// TIA Portal V16 program export: 1 tag tables, 0 data types, 1 data blocks, 2 code blocks (in call order from the OBs), 2 instance data blocks

VAR_GLOBAL   // PLC tag table "Default tag table"
   Clock_Byte AT %MB0 : Byte;
   Clock_10Hz AT %M0.0 : Bool;
   Clock_5Hz AT %M0.1 : Bool;
   "Clock_2.5Hz" AT %M0.2 : Bool;
   Clock_2Hz AT %M0.3 : Bool;
   "Clock_1.25Hz" AT %M0.4 : Bool;
   Clock_1Hz AT %M0.5 : Bool;
   "Clock_0.625Hz" AT %M0.6 : Bool;
   "Clock_0.5Hz" AT %M0.7 : Bool;
   "Disconect request" AT %M1.0 : Bool;
   "Send on/off" AT %M1.1 : Bool;
   "Receive enable" AT %M1.2 : Bool;
   "mine-tag" AT %M1.3 : Bool;
   nuevo_tag AT %M1.4 : Bool;
END_VAR

DATA_BLOCK "DATA"   // DB6
{ S7_Optimized_Access := 'TRUE' }
VERSION : 0.1
// stored: AutoNumber true, IsOnlyStoredInLoadMemory false, IsRetainMemResEnabled false, IsWriteProtectedInAS false, MemoryReserve 100
   VAR
      Receive : Array[0..20] of Char;
      Send : String := 'Hello world!';
      Do_Connect : Bool;
      Passive_Conn_Done : Bool;
   END_VAR
BEGIN
END_DATA_BLOCK

ORGANIZATION_BLOCK "Main"   // OB1, LAD, ProgramCycle
TITLE = "Main Program Sweep (Cycle)"
{ S7_Optimized_Access := 'TRUE' }
VERSION : 0.1
// stored: AutoNumber true, IsIECCheckEnabled false, SetENOAutomatically false
   VAR_INPUT
      Initial_Call : Bool;   // Initial call of this OB
      Remanence : Bool;   // =True, if remanent data are available
   END_VAR
   VAR_TEMP
      suma : Int;
   END_VAR
BEGIN

REGION Network 1
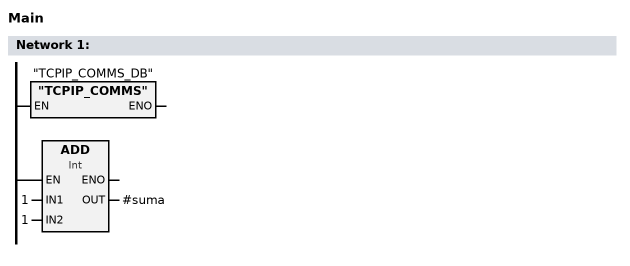
   RUNG wire#powerrail
      "TCPIP_COMMS_DB"()
   END_RUNG
   RUNG wire#powerrail
      { S7_Templates := "SrcType := Int" } Add(in1 := 1, in2 := 1, out => #suma)
   END_RUNG
   // the same network as SCL:
   "TCPIP_COMMS_DB"();   // "TCPIP_COMMS"
   #suma := 1 + 1;
END_REGION
END_ORGANIZATION_BLOCK

FUNCTION_BLOCK "TCPIP_COMMS"   // FB1, LAD
{ S7_Optimized_Access := 'TRUE' }
VERSION : 0.1
// stored: AutoNumber true, IsIECCheckEnabled false, IsRetainMemResEnabled false, MemoryReserve 100, SetENOAutomatically false, UDAEnableTagReadback false
   VAR
      TCON : Struct
         REQ : Bool;
         DONE : Bool;
         BUSY : Bool;
         ERROR : Bool;
         STATUS : UInt;
         DONESAVE : Bool;
      END_STRUCT;
      TDISCON : Struct
         REQ : Bool;
         DONE : Bool;
         BUSY : Bool;
         ERROR : Bool;
         DONESAVE : Bool;
         STATUS : UInt;
      END_STRUCT;
      TSEND : Struct
         REQ : Bool;
         DONE : Bool;
         BUSY : Bool;
         ERROR : Bool;
         DONESAVE : Bool;
         STATUS : UInt;
      END_STRUCT;
      TRCV : Struct
         EN_R : Bool;
         NDR : Bool;
         BUSY : Bool;
         ERROR : Bool;
         STATUS : UInt;
         RCVD_LEN : UDInt;
      END_STRUCT;
      ReceivedString : String;
      TCON_DB { ExternalAccessible := 'False'; ExternalVisible := 'False'; ExternalWritable := 'False'} : TCON;
      TDISCON_DB { ExternalAccessible := 'False'; ExternalVisible := 'False'; ExternalWritable := 'False'} : TDISCON;
      TSEND_DB { ExternalAccessible := 'False'; ExternalVisible := 'False'; ExternalWritable := 'False'} : TSEND;
      TRCV_DB { ExternalAccessible := 'False'; ExternalVisible := 'False'; ExternalWritable := 'False'} : TRCV;
   END_VAR
BEGIN

REGION Network 1: TCON
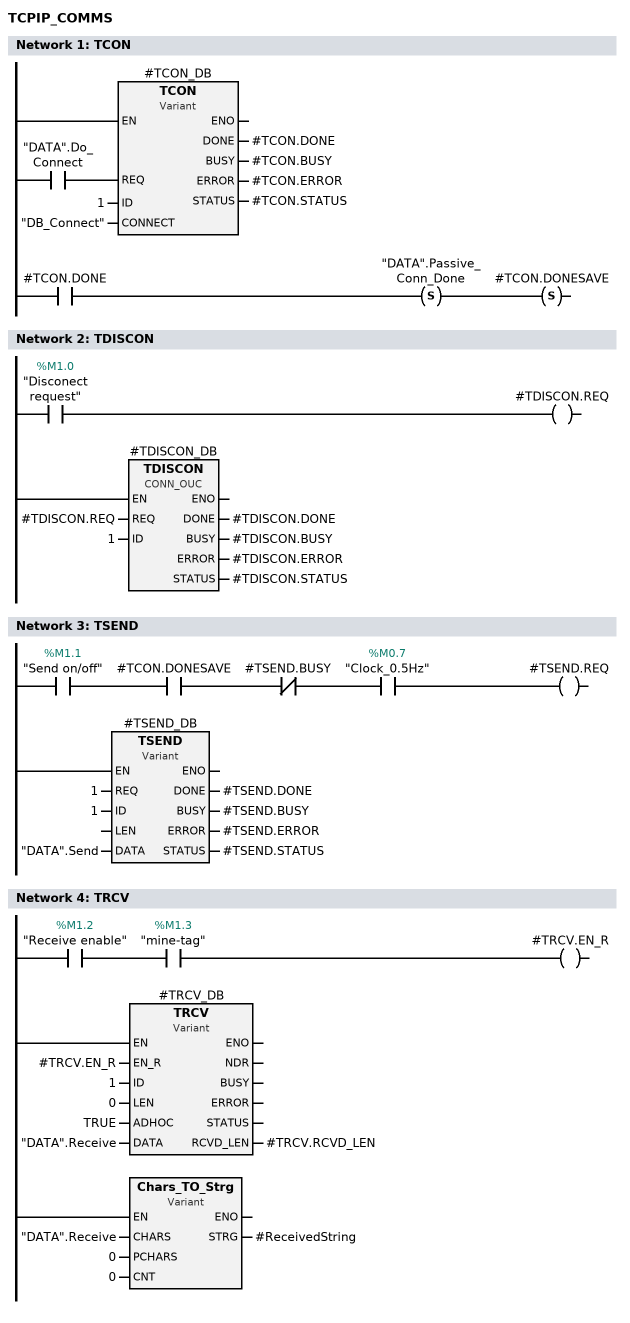
   RUNG wire#powerrail
      { S7_Templates := "[con_type := Variant, id_type := CONN_OUC]" } #TCON_DB.TCON(REQ := wire#w1, ID := 1, CONNECT := "DB_Connect", DONE => #TCON.DONE, BUSY => #TCON.BUSY, ERROR => #TCON.ERROR, STATUS => #TCON.STATUS)
   END_RUNG
   RUNG wire#powerrail
      Contact( "DATA".Do_Connect )
   END_RUNG wire#w1
   RUNG wire#powerrail
      Contact( #TCON.DONE )
      S_Coil( "DATA".Passive_Conn_Done )
      S_Coil( #TCON.DONESAVE )
   END_RUNG
   // the same network as SCL:
   #TCON_DB(REQ := "DATA".Do_Connect,   // TCON
            ID := 1,
            CONNECT := "DB_Connect",
            DONE => #TCON.DONE,
            BUSY => #TCON.BUSY,
            ERROR => #TCON.ERROR,
            STATUS => #TCON.STATUS);
   IF #TCON.DONE THEN
       "DATA".Passive_Conn_Done := TRUE;
       #TCON.DONESAVE := TRUE;
   END_IF;
END_REGION

REGION Network 2: TDISCON
   RUNG wire#powerrail
      Contact( "Disconect request" )
      Coil( #TDISCON.REQ )
   END_RUNG
   RUNG wire#powerrail
      { S7_Templates := "id_type := CONN_OUC" } #TDISCON_DB.TDISCON(REQ := #TDISCON.REQ, ID := 1, DONE => #TDISCON.DONE, BUSY => #TDISCON.BUSY, ERROR => #TDISCON.ERROR, STATUS => #TDISCON.STATUS)
   END_RUNG
   // the same network as SCL:
   #TDISCON.REQ := "Disconect request";
   #TDISCON_DB(REQ := #TDISCON.REQ,   // TDISCON
               ID := 1,
               DONE => #TDISCON.DONE,
               BUSY => #TDISCON.BUSY,
               ERROR => #TDISCON.ERROR,
               STATUS => #TDISCON.STATUS);
END_REGION

REGION Network 3: TSEND
   RUNG wire#powerrail
      Contact( "Send on/off" )
      Contact( #TCON.DONESAVE )
      I_Contact( #TSEND.BUSY )
      Contact( "Clock_0.5Hz" )
      Coil( #TSEND.REQ )
   END_RUNG
   RUNG wire#powerrail
      { S7_Templates := "[data_type := Variant, len_type := UDInt, id_type := CONN_OUC]" } #TSEND_DB.TSEND(REQ := 1, ID := 1, LEN :=, DATA := "DATA".Send, DONE => #TSEND.DONE, BUSY => #TSEND.BUSY, ERROR => #TSEND.ERROR, STATUS => #TSEND.STATUS)
   END_RUNG
   // the same network as SCL:
   #TSEND.REQ := "Send on/off" AND #TCON.DONESAVE AND NOT #TSEND.BUSY AND "Clock_0.5Hz";
   #TSEND_DB(REQ := 1,   // TSEND
             ID := 1,
             DATA := "DATA".Send,
             DONE => #TSEND.DONE,
             BUSY => #TSEND.BUSY,
             ERROR => #TSEND.ERROR,
             STATUS => #TSEND.STATUS);
END_REGION

REGION Network 4: TRCV
   RUNG wire#powerrail
      Contact( "Receive enable" )
      Contact( "mine-tag" )
      Coil( #TRCV.EN_R )
   END_RUNG
   RUNG wire#powerrail
      { S7_Templates := "[card := 1, ptr_type := Variant, value_type := UDInt, id_type := CONN_OUC]" } #TRCV_DB.TRCV(EN_R := #TRCV.EN_R, ID := 1, LEN := 0, ADHOC := TRUE, DATA := "DATA".Receive, NDR =>, BUSY =>, ERROR =>, STATUS =>, RCVD_LEN => #TRCV.RCVD_LEN)
   END_RUNG
   RUNG wire#powerrail
      { S7_Templates := "[ptr_type := Variant, str_type := String]" } Chars_TO_Strg(Chars := "DATA".Receive, pChars := 0, Cnt := 0, Strg => #ReceivedString)
   END_RUNG
   // the same network as SCL:
   #TRCV.EN_R := "Receive enable" AND "mine-tag";
   #TRCV_DB(EN_R := #TRCV.EN_R,   // TRCV
            ID := 1,
            LEN := 0,
            ADHOC := TRUE,
            DATA := "DATA".Receive,
            RCVD_LEN => #TRCV.RCVD_LEN);
   Chars_TO_Strg(Chars := "DATA".Receive, pChars := 0, Cnt := 0, Strg => #ReceivedString);
END_REGION
END_FUNCTION_BLOCK

DATA_BLOCK "TCPIP_COMMS_DB"   // DB1
VERSION : 0.1
// stored: AutoNumber true, InstanceOfName TCPIP_COMMS, InstanceOfType FB
"TCPIP_COMMS"
BEGIN
END_DATA_BLOCK

DATA_BLOCK "DB_Connect"   // DB2
{ S7_Optimized_Access := 'TRUE' }
// stored: AutoNumber true, InstanceOfName TCON_IP_v4, OfSystemLibElement TCON_IP_v4, OfSystemLibVersion 1.0
"TCON_IP_v4"
   // VAR
   //    InterfaceId : HW_ANY := 64;
   //    ID : CONN_OUC := 1;
   //    ConnectionType : Byte;
   //    ActiveEstablished : Bool := false;
   //    RemoteAddress { S7_SetPoint := 'True'} : IP_V4;
   //    RemotePort : UInt := 0;
   //    LocalPort : UInt := 5000;
   // END_VAR
BEGIN
   RemoteAddress.ADDR[1] := 192;
   RemoteAddress.ADDR[2] := 168;
   RemoteAddress.ADDR[3] := 1;
   RemoteAddress.ADDR[4] := 43;
END_DATA_BLOCK
